// Provides logger
INTERFACE I_Logger

// Logs the message without any additions.
METHOD LogDefault
VAR_INPUT
	message	: Tc2_System.T_MaxString;
END_VAR
END_METHOD

// Logs the message by adding the error header to the start.
METHOD LogError
VAR_INPUT
	message	: Tc2_System.T_MaxString;
END_VAR
END_METHOD

// Logs the message by adding the info header to the start.
METHOD LogInfo
VAR_INPUT
	message	: Tc2_System.T_MaxString;
END_VAR
END_METHOD

// Logs the message by adding the info header to the start.
METHOD LogWarning
VAR_INPUT
	message	: Tc2_System.T_MaxString;
END_VAR
END_METHOD

METHOD Reset
VAR_INPUT
END_VAR
END_METHOD

END_INTERFACE

(* stored: Version 1.1.0.1, ProductVersion 3.1.4024.14
   Itf I_Logger: Id {d290d270-2ea5-0094-355e-e10a816b0b83}
   Method LogDefault: Id {ab048765-d20e-0519-16de-3386aa7aef2d}
   Method LogError: Id {1c17d66c-c958-0bab-3657-7abaf0df7a63}
   Method LogInfo: Id {2a4bd426-acf4-0216-32e4-7a77254dddba}
   Method LogWarning: Id {cd7242be-bc18-041d-0fec-fd1ac71a6a27}
   Method Reset: Id {66b5eb65-53fe-0218-0604-9a9b8f46d191} *)
